  994 = 'S4_Prompts Default 994' | German: 'S4_Prompts German 994' | French: 'S4_Prompts French 994'
  995 = 'S4_Prompts Default 995' | German: 'S4_Prompts German 995' | French: 'S4_Prompts French 995'
  996 = 'S4_Prompts Default 996' | German: 'S4_Prompts German 996' | French: 'S4_Prompts French 996'
  997 = 'S4_Prompts Default 997' | German: 'S4_Prompts German 997' | French: 'S4_Prompts French 997'
  998 = 'S4_Prompts Default 998' | German: 'S4_Prompts German 998' | French: 'S4_Prompts French 998'
  999 = 'S4_Prompts Default 999' | German: 'S4_Prompts German 999' | French: 'S4_Prompts French 999'
  1000 = 'S4_Prompts Default 1000' | German: 'S4_Prompts German 1000' | French: 'S4_Prompts French 1000'
   = ''
END_TEXTLIST

(* stored: Version 1.1.0.1, ProductVersion 3.1.4024.12
   TextList S4_Prompts: Id {31f411e5-51a5-488a-9c18-48d2c22bfc30} *)
